{attribute 'GeneratedUsingTerminal: KL9900-0060'}
{attribute addProperty BoxType "KL9900-0060"}
{attribute addProperty Id "Channel_1AT %Q*Channel_7D202F580"}
{attribute addProperty CRC "1764799410"}
{attribute addProperty Size "0"}
TYPE KL_6930B3B2 :
STRUCT
	{attribute addProperty Name "Channel_1"}
	Channel_1 : Channel_7D202F58;
END_STRUCT
END_TYPE

(* stored: Version 1.2.0.0, ProductVersion 3.1.4024.9
   DUT KL_6930B3B2: Id {374e67de-5428-469b-a40c-c043eb478652} *)
